FUNCTION_BLOCK EBM_Power
VAR_INPUT
	EN: BOOL;
	ModbusRTU: REFERENCE TO ModbusRTU;
	Address: BYTE := 101;
END_VAR
VAR_OUTPUT
	ENO: BOOL;
	Power: LREAL;
END_VAR
VAR
	ModbusWord_T_Power: ModbusReadWord;
	ModbusWord_T_RefU: ModbusReadWord;
	ModbusWord_T_RefI: ModbusReadWord;
	T_RefU: LREAL;
	T_RefI: LREAL;
END_VAR
VAR // added by the converter: edge detectors and wires of the graphical bodies
    _w1, _w2, _w4, _w5 : ANY;
    _w3 : LREAL;
END_VAR

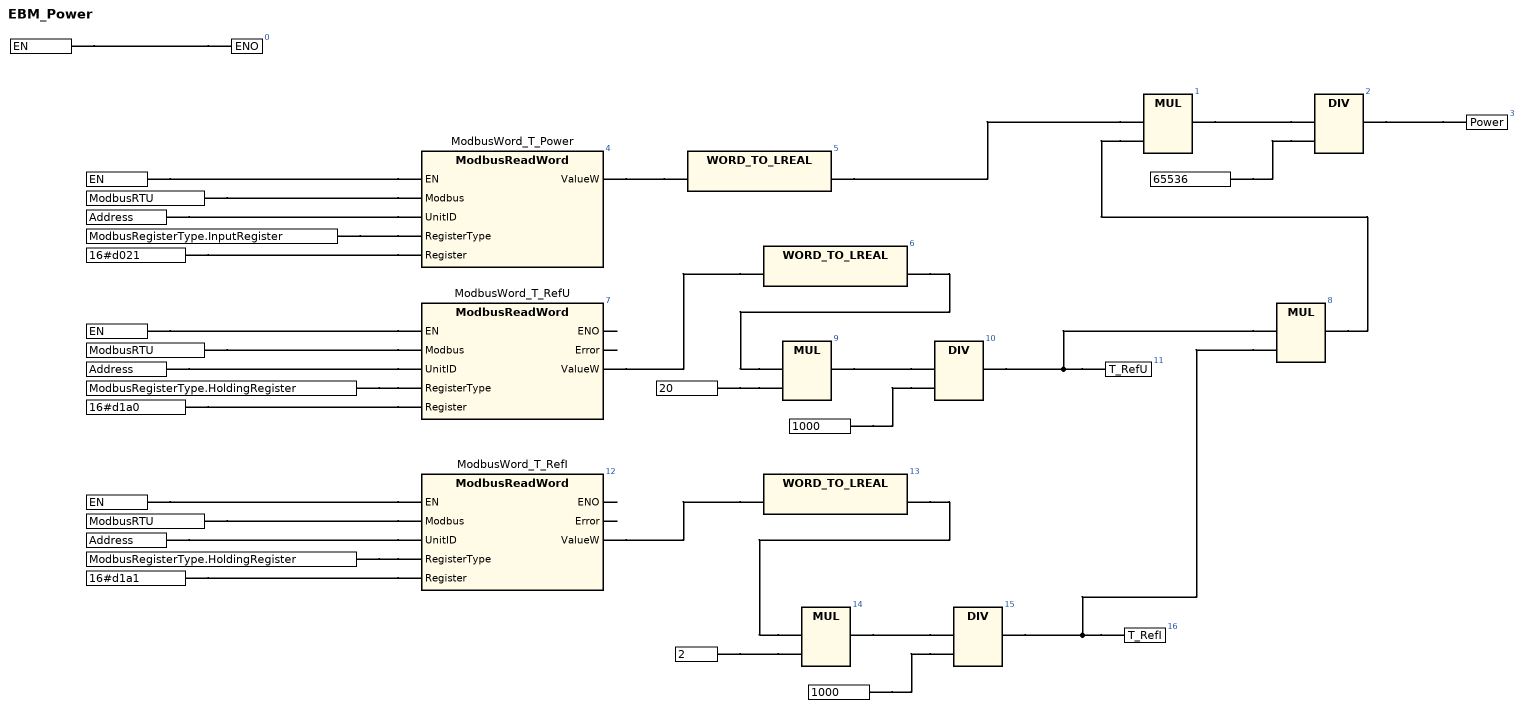
ENO := EN;
Power := (_w1 * _w2) / 65536;
ModbusWord_T_Power(
    EN := EN,
    Modbus := ModbusRTU,
    UnitID := Address,
    RegisterType := ModbusRegisterType.InputRegister,
    Register := 16#d021); // ModbusReadWord
_w1 := WORD_TO_LREAL(ModbusWord_T_Power.ValueW);
_w3 := WORD_TO_LREAL(ModbusWord_T_RefU.ValueW);
ModbusWord_T_RefU(
    EN := EN,
    Modbus := ModbusRTU,
    UnitID := Address,
    RegisterType := ModbusRegisterType.HoldingRegister,
    Register := 16#d1a0); // ModbusReadWord
_w2 := _w4 * _w5;
_w4 := (_w3 * 20) / 1000;
T_RefU := _w4;
ModbusWord_T_RefI(
    EN := EN,
    Modbus := ModbusRTU,
    UnitID := Address,
    RegisterType := ModbusRegisterType.HoldingRegister,
    Register := 16#d1a1); // ModbusReadWord
_w5 := (WORD_TO_LREAL(ModbusWord_T_RefI.ValueW) * 2) / 1000;
T_RefI := _w5;

END_FUNCTION_BLOCK

(* stored: Version 1.1.0.1, ProductVersion 3.1.4024.6
   POU EBM_Power: Id {0939ef26-dd0c-422b-ba4d-083ba3778d73}, SpecialFunc None *)
